{attribute 'GeneratedUsingTerminal: EL2595-0000-0019'}
{attribute addProperty BoxType "EL2595-0000-0019"}
{attribute addProperty Id "DOX_StatusAT %I*DOX_Status_F52B34D37DOX_ControlAT %Q*DOX_Control_75D5C9E23WcStateAT %I*WcState_9091E0EB2InfoDataAT %I*InfoData_94A18F5E2"}
{attribute addProperty CRC "2494939881"}
{attribute addProperty Size "14"}
TYPE EL2595_94B5C2E9 EXTENDS EtcSlaveTerminalBase_947E5A46 :
STRUCT
	{attribute addProperty Name "DOX_Status"}
	DOX_Status : DOX_Status_F52B34D3;
	{attribute addProperty Name "DOX_Control"}
	DOX_Control : DOX_Control_75D5C9E2;
	{attribute addProperty Name "WcState"}
	WcState : WcState_9091E0EB;
	{attribute addProperty Name "InfoData"}
	InfoData : InfoData_94A18F5E;
END_STRUCT
END_TYPE

(* stored: Version 1.2.0.0, ProductVersion 3.1.4024.9
   DUT EL2595_94B5C2E9: Id {a212aaf2-a340-40ef-9d3e-1000f561fae3} *)
